FUNCTION_BLOCK "FC9000"
{ S7_Optimized_Access := 'TRUE' }
VERSION : 0.1

BEGIN
	(*some changes*)
	(*some changes again!*)
END_FUNCTION_BLOCK

